TYPE E_FunctionType :
(**************************************************************************************
 * 	Application		:	BoxControl Framework
 *	Revision		:	$Revision: 404529 $
 *	Revision date	:	$Date: 2018-04-23 08:21:38 +0200 (Mo., 23 Apr 2018) $
 *	Last changed by	:	$Author: b7bolm $
 *	URL				:	$URL: http://almscdc.swisslog.com/repo/SWPD/Development/BoxControlFramework/20_Release/trunk/01_Software/BCF/BCF/JumpStart/20_Product/10_App/12_E_Functions/10_Lib/10_Conv/01_DUTs/E_FunctionType.TcDUT $
 *
 *	Purpose			:	Function type definition
 *
 * ------------------------------------------------------------------------------------
 *	Copyright Swisslog [IP AG], Switzerland. All rights reserved.
 * 
 * ------------------------------------------------------------------------------------
 *	
 * 	Revision History: 
 *
 * 	VERSION			DATE			INITIALS			DESCRIPTION
 *	0.1				01.01.2001		swl					Example
 *
 **************************************************************************************)	
(
	NO_TYPE,
	Scanner
);
END_TYPE

(* stored: Version 1.1.0.1, ProductVersion 3.1.4024.9
   DUT E_FunctionType: Id {c15d865c-b37f-4260-8c78-43913a1f5a57} *)
